Fanuc KAREL source: NC0028.KL

-- PROVISIONAL review KL for V940-1; original PC SHA256 7058c5d0af4d3c048d7ec84ec6ff4a0afbf33adf3cee1307d08eea303c7aab6d
-- Incomplete behavior may be omitted. Consult companion uncertainty JSON. Do not deploy.
PROGRAM NC0028
%NOLOCKGROUP
-- UNRESOLVED_LOCAL_POOL 1 cells at code offset 3; source declarations unknown
-- DIRECT_LOCAL_WORD_ACCESS alone does not prove INTEGER, REAL, or BOOLEAN
BEGIN
  -- UNRESOLVED_PC offsets 0-8; opcodes 2B,2C,7B
  -- UNRESOLVED_PC offsets 13-20; opcodes 9D,23
  -- UNRESOLVED_PC offsets 25-42; opcodes 21,40,41,42
  -- UNRESOLVED_PC offsets 47-64; opcodes 21,40,41,42
  -- UNRESOLVED_PC offsets 69-86; opcodes 21,40,41,42
  -- UNRESOLVED_PC offsets 91-108; opcodes 21,40,41,42
  -- UNRESOLVED_PC offsets 113-130; opcodes 21,40,41,42
  -- UNRESOLVED_PC offsets 135-152; opcodes 21,40,41,42
  -- UNRESOLVED_PC offsets 157-174; opcodes 21,40,41,42
  -- UNRESOLVED_PC offsets 179-196; opcodes 21,40,41,42
  -- UNRESOLVED_PC offsets 201-218; opcodes 21,40,41,42
  -- UNRESOLVED_PC offsets 223-240; opcodes 21,40,41,42
  -- UNRESOLVED_PC offsets 245-262; opcodes 21,40,41,42
  -- UNRESOLVED_PC offsets 267-284; opcodes 21,40,41,42
  -- UNRESOLVED_PC offsets 289-319; opcodes 21,9D,52,23,7A,40,41,42
  -- UNRESOLVED_PC offsets 324-348; opcodes 21,2E,52,23,7A,43
  -- UNRESOLVED_PC offsets 353-371; opcodes 21,2E,52,23
  -- UNRESOLVED_PC offsets 376-392; opcodes 7A,40,41,42
  -- UNRESOLVED_PC offsets 397-421; opcodes 21,2E,52,23,7A,43
  -- UNRESOLVED_PC offsets 426-444; opcodes 21,2E,52,23
  -- UNRESOLVED_PC offsets 449-465; opcodes 7A,40,41,42
  -- UNRESOLVED_PC offsets 470-494; opcodes 21,2E,52,23,7A,43
  -- UNRESOLVED_PC offsets 499-517; opcodes 21,2E,52,23
  -- UNRESOLVED_PC offsets 522-538; opcodes 7A,40,41,42
  -- UNRESOLVED_PC offsets 543-567; opcodes 21,2E,52,23,7A,43
  -- UNRESOLVED_PC offsets 572-590; opcodes 21,2E,52,23
  -- UNRESOLVED_PC offsets 595-611; opcodes 7A,40,41,42
  -- UNRESOLVED_PC offsets 616-640; opcodes 21,2E,52,23,7A,43
  -- UNRESOLVED_PC offsets 645-663; opcodes 21,2E,52,23
  -- UNRESOLVED_PC offsets 668-684; opcodes 7A,40,41,42
  -- UNRESOLVED_PC offsets 689-713; opcodes 21,2E,52,23,7A,43
  -- UNRESOLVED_PC offsets 718-736; opcodes 21,2E,52,23
  -- UNRESOLVED_PC offsets 741-757; opcodes 7A,40,41,42
  -- UNRESOLVED_PC offsets 762-786; opcodes 21,2E,52,23,7A,43
  -- UNRESOLVED_PC offsets 791-809; opcodes 21,2E,52,23
  -- UNRESOLVED_PC offsets 814-830; opcodes 7A,40,41,42
  -- UNRESOLVED_PC offsets 835-859; opcodes 21,2E,52,23,7A,43
  -- UNRESOLVED_PC offsets 864-882; opcodes 21,2E,52,23
  -- UNRESOLVED_PC offsets 887-903; opcodes 7A,40,41,42
  -- UNRESOLVED_PC offsets 908-932; opcodes 21,2E,52,23,7A,43
  -- UNRESOLVED_PC offsets 937-955; opcodes 21,2E,52,23
  -- UNRESOLVED_PC offsets 960-976; opcodes 7A,40,41,42
  -- UNRESOLVED_PC offsets 981-1005; opcodes 21,2E,52,23,7A,43
  -- UNRESOLVED_PC offsets 1010-1028; opcodes 21,2E,52,23
  -- UNRESOLVED_PC offsets 1033-1049; opcodes 7A,40,41,42
  -- UNRESOLVED_PC offsets 1054-1078; opcodes 21,2E,52,23,7A,43
  -- UNRESOLVED_PC offsets 1083-1101; opcodes 21,2E,52,23
  -- UNRESOLVED_PC offsets 1106-1122; opcodes 7A,40,41,42
  -- UNRESOLVED_PC offsets 1127-1151; opcodes 21,2E,52,23,7A,43
  -- UNRESOLVED_PC offsets 1156-1174; opcodes 21,2E,52,23
  -- UNRESOLVED_PC offsets 1184-1188; opcodes 7F
  -- UNRESOLVED_PC offsets 1193-1197; opcodes 27,AA
  -- UNRESOLVED_PC offsets 1202-1206; opcodes 7F
END NC0028
